Fanuc KAREL source: kc00045.KL

-- PROVISIONAL review KL for V940-1; original PC SHA256 d83fe0f54162c8294c68851acfa7a8500cfac93e0ef679a11a49049a5342da33
-- Incomplete behavior may be omitted. Consult companion uncertainty JSON. Do not deploy.
PROGRAM KC00045
%NOLOCKGROUP
BEGIN
  -- V9_ZERO_TABLE_METADATA_HINT layout=0002_ascii; no indexed target words; source/name/runtime held
  -- UNRESOLVED_PC offsets 5-29; opcodes 27,22,22,2A,22,31
  -- UNRESOLVED_PC offsets 34-38; opcodes 7F
END KC00045
